{attribute 'qualified_only'}
VAR_GLOBAL
	

err_ack		AT %Q*	:	BOOL;
run			AT %Q*	:	BOOL;

bEstopSet	AT %I*	:	BOOL;

END_VAR

(* stored: Version 1.1.0.1, ProductVersion 3.1.4024.12
   GVL SAFETY: Id {2263d95c-9ada-478e-aa68-a737c3d0fac6} *)
